# EPICS substitutions: db/Beckhoff_3XXX/ecmcEL3702.substitutions
file "ecmcEcSlave.template"
{
  pattern {}
          {}
}

file "ecmcEL37XX-chX.template"
{
  pattern {CH_ID, DTYP,             FTVL  }
          {1,     asynInt16ArrayIn, SHORT }
          {2,     asynInt16ArrayIn, SHORT }
}
